FUNCTION_BLOCK FB_Uitmalen
VAR_INPUT
	
END_VAR
VAR_OUTPUT
END_VAR
VAR
	stap : INT;
	offPomp : E_POMPSTATE :=E_POMPSTATE.off;
	standbyRegelschuif : E_RegelschuifState := E_RegelschuifState.standby;
	closed : E_OpenDichtKlepState :=E_OpenDichtKlepState.closed;
	open : E_OpenDichtKlepState :=E_OpenDichtKlepState.open;
	//toerentaltotaal 
	optoeren : E_PompState :=E_PompState.optoeren;
	
	CurrentModus : E_Besturingsmodus;
	KlepV2012 : ITF_OpenDichtKlep;
	KlepV2014 : ITF_OpenDichtKlep;
	KlepV2021 : ITF_OpenDichtKlep;
	KlepV2023 : ITF_OpenDichtKlep;
	KlepV2024 : ITF_OpenDichtKlep;
	KlepV2025 : ITF_OpenDichtKlep;
	KlepV2026 : ITF_OpenDichtKlep;
	
	
	SchuifV2013_AFG : ITF_Regelschuif;
	SchuifV2022_AFG : ITF_Regelschuif;
	
	SchuifV2013_DG : ITF_Regelschuif;
	SchuifV2022_DG : ITF_Regelschuif;
	
	Pomp1_P2011 : ITF_Pomp;
	pomp2_P2021 : ITF_Pomp;
	
	pompP2011:INT;
	pompP2021:INT;
END_VAR

currentmodus := main.Regelingen.BestuurMode;
IF currentmodus = E_Besturingsmodus.uitmalen THEN	
CASE stap OF
	1:
		Pomp1_P2011.PompGoTo(0);
		pomp2_P2021.PompGoTo(0);
		IF 0 = Pomp1_P2011.ActueelToerental  AND offPomp = Pomp1_P2011.StatePomp AND 0 = pomp2_P2021.ActueelToerental  AND offPomp = pomp2_P2021.StatePomp THEN
			stap := 2;
		END_IF
			
	2:
		SchuifV2013_AFG.RegelschuifGoTo(0);
		SchuifV2022_AFG.RegelschuifGoTo(0);
		KlepV2014.Close();
		KlepV2021.Close();
		KlepV2024.Close();
		KlepV2026.Close();
		IF 0 = SchuifV2013_AFG.ActueelPosition  AND standbyRegelschuif = SchuifV2013_AFG.StateRegelschuif AND  0 = SchuifV2022_AFG.ActueelPosition  AND standbyRegelschuif = SchuifV2022_AFG.StateRegelschuif AND closed = KlepV2014.StateKlep AND closed = KlepV2021.StateKlep AND  closed = KlepV2024.StateKlep  AND  closed = KlepV2026.StateKlep  THEN
			stap := 3;
		END_IF
	3:
		// totaal toerental
		pompP2011 := main.Regelingen.ToerentalP2011; // get toerental 11
		pompP2021 := main.Regelingen.ToerentalP2021; // get toerental 21
		pomp2_P2021.PompGoTo(pompP2021);//Set toerental 21
		Pomp1_P2011.PompGoTo(pompP2011); // set toerental 11
		
		
		IF optoeren = Pomp1_P2011.StatePomp THEN 
			KlepV2012.Open();
			IF open = KlepV2012.StateKlep THEN
				KlepV2012.Close();
			END_IF
		END_IF
		
		IF optoeren = pomp2_P2021.StatePomp THEN 
			KlepV2021.Open();
			KlepV2024.Open();
			IF open = KlepV2021.StateKlep AND open = KlepV2024.StateKlep THEN
				KlepV2021.Close();
				KlepV2024.Close();
			END_IF
		END_IF
		
END_CASE
END_IF

//FB_Init is always available implicitly and it is used primarily for initialization.
//The return value is not evaluated. For a specific influence, you can also declare the
//methods explicitly and provide additional code there with the standard initialization
//code. You can evaluate the return value.
METHOD FB_Init: BOOL
VAR_INPUT
    bInitRetains: BOOL; // TRUE: the retain variables are initialized (reset warm / reset cold)
    bInCopyCode: BOOL;  // TRUE: the instance will be copied to the copy code afterward (online change)   
		OpenDichtKlepV2012: ITF_OpenDichtKlep;
	OpenDichtKlepV2014: ITF_OpenDichtKlep;
	OpenDichtKlepV2021: ITF_OpenDichtKlep;
	OpenDichtKlepV2023: ITF_OpenDichtKlep;
	OpenDichtKlepV2024: ITF_OpenDichtKlep;
	OpenDichtKlepV2025: ITF_OpenDichtKlep;
	OpenDichtKlepV2026: ITF_OpenDichtKlep;

	RegelschuifV2013_AFO: ITF_Regelschuif;
	RegelschuifV2022_AFO: ITF_Regelschuif;
	
	PompP2021: ITF_Pomp;
	PompP2011: ITF_Pomp;


	RegelschuifV2013_DG: ITF_Regelschuif;
	RegelschuifV2022_DG: ITF_Regelschuif;
END_VAR

	
KlepV2012 := OpenDichtKlepV2012;
KlepV2014 := OpenDichtKlepV2014;
KlepV2021 := OpenDichtKlepV2021;
KlepV2023 := OpenDichtKlepV2023;
KlepV2024 := OpenDichtKlepV2024;
KlepV2025 := OpenDichtKlepV2025;
KlepV2026 := OpenDichtKlepV2026;

SchuifV2013_AFG := RegelschuifV2013_AFO;
SchuifV2022_AFG := RegelschuifV2022_AFO;
SchuifV2013_DG := RegelschuifV2013_DG;
SchuifV2022_DG := RegelschuifV2022_DG;

pomp2_P2021 := PompP2021;
pomp1_p2011 := PompP2011;
END_METHOD

END_FUNCTION_BLOCK

(* stored: Version 1.1.0.1, ProductVersion 3.1.4026.8
   POU FB_Uitmalen: Id {9ae4d82e-20f8-4e09-9aaa-bd1ddcd0f3cd}, SpecialFunc None
   Method FB_Init: Id {f1bb211c-677d-41cb-9dca-60535f7173bb} *)
